FUNCTION f_Subtraction : REAL
VAR_INPUT
	rDiff1	:	REAL;
	rDiff2	:	REAL;
END_VAR
VAR
END_VAR

f_Subtraction := rDiff1 - rDiff2;

END_FUNCTION

(* stored: Version 1.1.0.1, ProductVersion 3.1.4024.12
   POU f_Subtraction: Id {454c2c90-4657-401d-846b-fbc6db92f524}, SpecialFunc None *)
